TYPE ST_Configuration :
STRUCT
  XtsStationParameter  : ARRAY[1..MAX_STATION] OF ST_STATION_PARAMETER;
END_STRUCT
END_TYPE

(* stored: Version 1.1.0.1, ProductVersion 3.1.4024.13
   DUT ST_Configuration: Id {751e9be0-0116-4a27-b9d5-2088d21242fd} *)
